// TIA Portal V19 export
DATA_BLOCK "Alarm_No2"   // DB7
// stored: InstanceOfName Alarm_Trigger, InstanceOfType FB
"Alarm_Trigger"
   // VAR_INPUT
   //    Alarm_Trigger : Bool;
   //    Timer_PT : Time;
   //    Ack_PB : Bool;
   //    Reset_PB : Bool;
   // END_VAR
   // VAR_OUTPUT
   //    ALARM : Bool;
   //    ALARM_ACKED : Bool;
   //    ALARM_BLINK : Bool;
   // END_VAR
   // VAR
   //    Alarm_TD : Bool;
   //    Alarm_Active : Bool;
   //    Alarm_ACK : Bool;
   //    Alarm_Reset : Bool;
   //    Alarm_Timer { S7_SetPoint := 'True'} : TON_TIME;
   // END_VAR
BEGIN
END_DATA_BLOCK
